{attribute 'qualified_only'}
{attribute 'strict'}
TYPE E_CAMERA_Vendor :
(
	SIEMENS		:= 1,
	OMRON 		:= 2,
	KEYENCE		:= 3,
	COGNEX		:= 4,
	HIKROBOT	:= 5
);
END_TYPE

(* stored: Version 1.1.0.1
   DUT E_CAMERA_Vendor: Id {b685a197-480d-4fe9-b238-5737b7c6ed26} *)
